(* IEC 61131-3 sources: SemaPLC/sema-plc-web/templates/.sema/skills/plc-build-and-verify/st-patterns, 6 files *)

(* ---- bangbang_plant.st ---- *)
(* 模式:双位(bang-bang)回差控制 + 自驱 plant(水箱/温控通用骨架)
   核心:液位低于 LOW 开阀,高于 HIGH 关阀,中间保持(回差防频繁切换)。
   plant 模型:开阀时液位升、关阀时降,饱和到 [0, 1000]。
   改写要点:
   - 改 LOW/HIGH 阈值
   - 改 plant 动态(升降速率、是否有恒定泄漏)
   - 温控场景:valve→heater, level→temperature, 降=自然散热 *)
PROGRAM tank_bangbang
  VAR
    level AT %QW0 : INT;            (* 当前液位:自驱量,仿真绑它 *)
    inlet_valve AT %QX0.0 : BOOL;   (* 进水阀开关 *)
  END_VAR
  VAR
    LOW : INT := 200;               (* 下限阈值 *)
    HIGH : INT := 800;              (* 上限阈值 *)
  END_VAR

  (* 回差逻辑:低于下限开、高于上限关、中间保持上一状态 *)
  IF level < LOW THEN
    inlet_valve := TRUE;
  ELSIF level > HIGH THEN
    inlet_valve := FALSE;
  END_IF;

  (* === plant 模型(自驱,仿真能动的关键)=== *)
  IF inlet_valve THEN
    level := level + 5;             (* 开阀:每周期升 5 *)
  ELSE
    level := level - 3;             (* 关阀:自然泄漏降 3 *)
  END_IF;

  (* 饱和 *)
  IF level > 1000 THEN level := 1000; END_IF;
  IF level < 0 THEN level := 0; END_IF;
END_PROGRAM

CONFIGURATION Config0
  RESOURCE Res0 ON PLC
    TASK Main(INTERVAL := T#50ms, PRIORITY := 0);
    PROGRAM Inst0 WITH Main : tank_bangbang;
  END_RESOURCE
END_CONFIGURATION

(* ---- conveyor_shift_register.st ---- *)
(* 模式:传送带工件追踪 + 移位寄存器分拣(最难场景骨架)
   验证纪律(关键):移位寄存器单脉冲几个周期就移走,任何采样都追不上——
   verify 时用 steady+pulseScans 投一个干净脉冲,断言它【留下的持久后果】
   (推杆锁存 / 计数 +1),别设计逐格追 bit 的工况。
   仿真:工件位置 wp_pos 是内部自驱量(随带走),translateX 绑它。
   改写要点:改料道数、传感器位置阈值、SLOTS 长度 *)
PROGRAM conveyor_sort
  VAR
    belt_run AT %IX0.0 : BOOL;        (* 启动传送带 *)
    color_sensor AT %IX0.1 : BOOL;    (* 入口颜色/检测传感器(脉冲)*)
    wp_pos AT %QW0 : INT;             (* 工件位置 0-1000:自驱量,仿真 translateX 绑它 *)
    pusher1 AT %QX0.0 : BOOL;         (* 料道1推杆 *)
    sort_count AT %QW1 : INT;         (* 已分拣计数 *)
  END_VAR
  VAR
    sensor_edge : R_TRIG;
    item_on_belt : BOOL := FALSE;     (* 带上有工件(锁存)*)
    push_latch : TON;                 (* 推杆动作保持 *)
  END_VAR

  sensor_edge(CLK := color_sensor);

  (* 入口检测到工件 → 锁存"带上有工件",位置归零开始走 *)
  IF sensor_edge.Q AND NOT item_on_belt THEN
    item_on_belt := TRUE;
    wp_pos := 0;
  END_IF;

  (* === plant:工件随带前进(自驱量,仿真动画的关键)=== *)
  IF belt_run AND item_on_belt THEN
    wp_pos := wp_pos + 10;
  END_IF;

  (* 到达料道1工位(阈值 500)→ 触发推杆 + 计数 +1(持久后果)*)
  IF item_on_belt AND wp_pos >= 500 THEN
    push_latch(IN := TRUE, PT := T#500ms);
    pusher1 := TRUE;
    IF wp_pos >= 510 AND wp_pos <= 520 THEN   (* 只在跨过工位的那一刻计数一次 *)
      sort_count := sort_count + 1;
    END_IF;
  END_IF;

  (* 工件走到带尾 → 复位,等下一个 *)
  IF wp_pos >= 1000 THEN
    item_on_belt := FALSE;
    pusher1 := FALSE;
    push_latch(IN := FALSE);
  END_IF;
END_PROGRAM

CONFIGURATION Config0
  RESOURCE Res0 ON PLC
    TASK Main(INTERVAL := T#50ms, PRIORITY := 0);
    PROGRAM Inst0 WITH Main : conveyor_sort;
  END_RESOURCE
END_CONFIGURATION

(* ---- edge_counter.st ---- *)
(* 模式:R_TRIG 边沿计数 + 下限钳位 + 阈值比较输出(停车场/产线计数通用骨架)
   核心:两个 R_TRIG 分别取入口/出口上升沿,驱动 INT 加/减,
   与上限比较控制 BOOL 输出(满位灯/闸机)。
   改写要点:
   - 改传感器数量(单向计数只保留 entry_edge)
   - 改上限值(MAX_COUNT)
   - 加多级阈值(如 80% 预警灯) *)
PROGRAM parking_counter
  VAR
    entry_sensor AT %IX0.0 : BOOL;   (* 入口传感器 *)
    exit_sensor AT %IX0.1 : BOOL;    (* 出口传感器 *)
    car_count AT %QW0 : INT;         (* 当前车辆数 *)
    full_light AT %QX0.0 : BOOL;     (* 满位指示灯 *)
    gate_entry AT %QX0.1 : BOOL;     (* 入口闸机,TRUE=放行 *)
  END_VAR
  VAR
    entry_edge : R_TRIG;
    exit_edge : R_TRIG;
    MAX_COUNT : INT := 10;           (* 车位上限,按需改 *)
  END_VAR

  entry_edge(CLK := entry_sensor);
  exit_edge(CLK := exit_sensor);

  (* 加减计数,下限钳 0 *)
  IF entry_edge.Q THEN
    car_count := car_count + 1;
  END_IF;
  IF exit_edge.Q AND car_count > 0 THEN
    car_count := car_count - 1;
  END_IF;

  (* 阈值比较 → 输出 *)
  full_light := (car_count >= MAX_COUNT);
  gate_entry := (car_count < MAX_COUNT);
END_PROGRAM

CONFIGURATION Config0
  RESOURCE Res0 ON PLC
    TASK Main(INTERVAL := T#20ms, PRIORITY := 0);
    PROGRAM Inst0 WITH Main : parking_counter;
  END_RESOURCE
END_CONFIGURATION

(* ---- latch_priority.st ---- *)
(* 模式:输入驱动锁存 + 优先级覆盖(电机启停/阀门启停通用骨架)
   核心:motor := (start OR motor) AND NOT stop AND NOT estop
   急停/停止在 AND 链末端 → 天然最高优先(同时按下时停止必赢)。
   改写要点:
   - 改输入/输出名与数量
   - 多组互锁:复制锁存行,加互斥条件(如 motor1 AND NOT motor2)
   - 需要脉冲启动(按一下松开仍保持)时已内建——start 松开后 motor 自锁 *)
PROGRAM motor_latch
  VAR
    start_btn AT %IX0.0 : BOOL;   (* 启动按钮 *)
    stop_btn AT %IX0.1 : BOOL;    (* 停止按钮 *)
    estop AT %IX0.2 : BOOL;       (* 急停,优先级最高 *)
    motor AT %QX0.0 : BOOL;       (* 电机输出 *)
    run_light AT %QX0.1 : BOOL;   (* 运行指示灯 *)
  END_VAR

  (* 一行锁存:start 上升沿置位,stop/estop 随时复位;
     estop 在最外层 AND NOT → 即使 start 持续按住也能停 *)
  motor := (start_btn OR motor) AND NOT stop_btn AND NOT estop;
  run_light := motor;
END_PROGRAM

CONFIGURATION Config0
  RESOURCE Res0 ON PLC
    TASK Main(INTERVAL := T#20ms, PRIORITY := 0);
    PROGRAM Inst0 WITH Main : motor_latch;
  END_RESOURCE
END_CONFIGURATION

(* ---- pid_level_with_plant.st ---- *)
(* 模式:连续量闭环 + 内部 plant 自驱(液位/温度/流量 PID 或比例通用)
   关键(S1 硬门要求):被仿真的连续量(level)必须是【程序自驱的内部量/输出】,
   不能是 %IW 外部输入——否则实时仿真里它恒为初值=死图。
   改写要点:
   - 设定值 setpoint 做成 %IW 输入(用户拖 slider 给)
   - 反馈量 level 是内部 plant:由阀门开度自驱(进>出则升,反之降),饱和到 [0,1000]
   - 仿真把 height 绑到 level(自驱量),slider 绑到 setpoint(%IW) *)
PROGRAM pid_level
  VAR
    setpoint AT %IW0 : INT;     (* 设定值 0-1000,用户 slider 驱动 *)
    valve AT %QW0 : INT;        (* 阀门开度输出 0-1000 *)
    level AT %QW1 : INT;        (* 液位:做成输出/自驱量,仿真绑它 *)
  END_VAR
  VAR
    err : INT;
    inflow : INT;
  END_VAR

  (* === 控制器:比例控制,阀门开度随偏差 === *)
  err := setpoint - level;
  IF err > 0 THEN
    valve := err * 2;           (* 偏差越大开越大;按需换成完整 PID *)
    IF valve > 1000 THEN valve := 1000; END_IF;
  ELSE
    valve := 0;
  END_IF;

  (* === plant 模型(自驱闭环,这段是仿真能动起来的关键)===
     进水正比阀门开度,出水恒定泄漏;液位 = 上次 + 进 - 出,饱和 *)
  inflow := valve / 100;        (* 阀全开每周期进 10 *)
  level := level + inflow - 3;  (* 恒定泄漏 3 *)
  IF level > 1000 THEN level := 1000; END_IF;
  IF level < 0 THEN level := 0; END_IF;
END_PROGRAM

CONFIGURATION Config0
  RESOURCE Res0 ON PLC
    TASK Main(INTERVAL := T#50ms, PRIORITY := 0);
    PROGRAM Inst0 WITH Main : pid_level;
  END_RESOURCE
END_CONFIGURATION

(* ---- state_machine_timed.st ---- *)
(* 模式:N 状态机 + TON 定时器(红绿灯/顺序动作通用骨架)
   改写要点:
   - 改 state 取值数与每态的输出映射、PT 时长
   - 倒计时量 countdown 自动从定时器派生,直接绑数显
   - 这是"离散状态机自驱",部署即自动循环,无需外部输入 *)
PROGRAM state_machine
  VAR
    (* 输出:按需改名/增减 *)
    out_a AT %QX0.0 : BOOL;
    out_b AT %QX0.1 : BOOL;
    out_c AT %QX0.2 : BOOL;
    countdown AT %QW0 : INT;
  END_VAR
  VAR
    state : INT := 0;          (* 0/1/2... 按需扩展 *)
    cnt : INT := 0;            (* 当前态剩余秒 *)
    phase_timer : TON;
    tick : R_TRIG;
  END_VAR

  (* 1Hz 自激节拍:timer.Q 每秒翻一次,R_TRIG 取上升沿 = 每秒一个 tick *)
  phase_timer(IN := NOT phase_timer.Q, PT := T#1s);
  tick(CLK := phase_timer.Q);

  (* 首扫描初始化当前态时长(避免 cnt 初值 0 直接跳态)*)
  IF state = 0 AND cnt = 0 THEN cnt := 3; END_IF;

  IF tick.Q THEN
    cnt := cnt - 1;
    IF cnt <= 0 THEN
      CASE state OF
        0: state := 1; cnt := 1;   (* 态0持续3s → 态1持续1s *)
        1: state := 2; cnt := 2;   (* 态1 → 态2持续2s *)
        2: state := 0; cnt := 3;   (* 态2 → 回态0 *)
      END_CASE;
    END_IF;
  END_IF;

  (* 输出映射:任一时刻只有一个有效(按需改)*)
  out_a := (state = 0);
  out_b := (state = 1);
  out_c := (state = 2);
  countdown := cnt;
END_PROGRAM

CONFIGURATION Config0
  RESOURCE Res0 ON PLC
    TASK Main(INTERVAL := T#20ms, PRIORITY := 0);
    PROGRAM Inst0 WITH Main : state_machine;
  END_RESOURCE
END_CONFIGURATION
